// TIA Portal V20 export
ORGANIZATION_BLOCK "MainOB"   // OB126, LAD, ProgramCycle
TITLE = "Main Program Sweep (Cycle)"
{ S7_Optimized_Access := 'TRUE' }
// stored: SetENOAutomatically false
   VAR_INPUT
      Initial_Call : Bool;   // Initial call of this OB
      Remanence : Bool;   // =True, if remanent data are available
   END_VAR
   VAR_TEMP
      Temp : Bool;
   END_VAR
   VAR CONSTANT
      Constant_1 : Bool;
   END_VAR
BEGIN

REGION Network 1
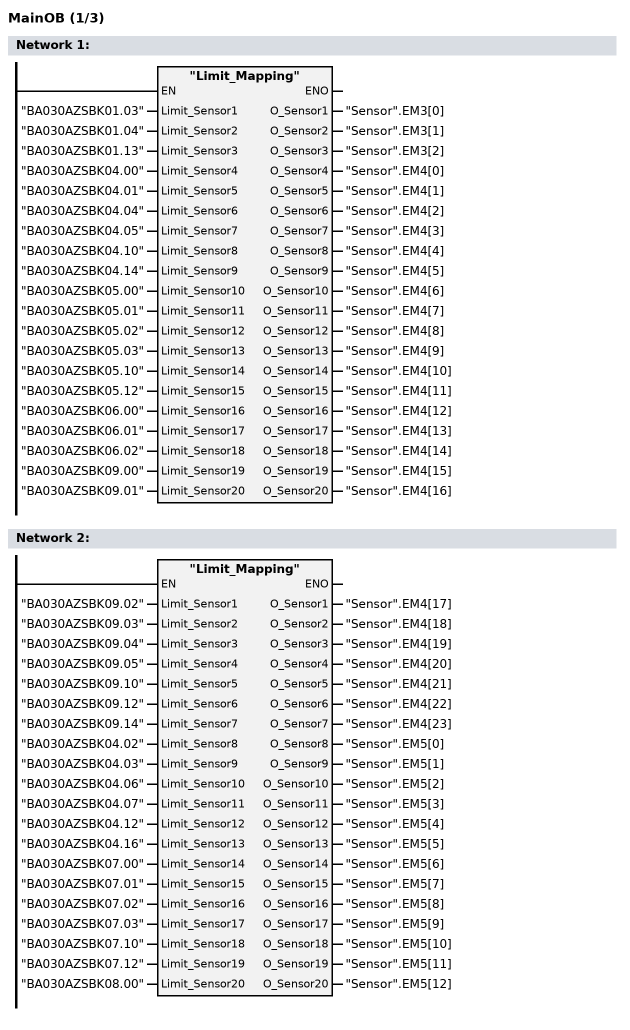
   RUNG wire#powerrail
      "Limit_Mapping"(Limit_Sensor1 := "BA030AZSBK01.03", Limit_Sensor2 := "BA030AZSBK01.04", Limit_Sensor3 := "BA030AZSBK01.13", Limit_Sensor4 := "BA030AZSBK04.00", Limit_Sensor5 := "BA030AZSBK04.01", Limit_Sensor6 := "BA030AZSBK04.04", Limit_Sensor7 := "BA030AZSBK04.05", Limit_Sensor8 := "BA030AZSBK04.10", Limit_Sensor9 := "BA030AZSBK04.14", Limit_Sensor10 := "BA030AZSBK05.00", Limit_Sensor11 := "BA030AZSBK05.01", Limit_Sensor12 := "BA030AZSBK05.02", Limit_Sensor13 := "BA030AZSBK05.03", Limit_Sensor14 := "BA030AZSBK05.10", Limit_Sensor15 := "BA030AZSBK05.12", Limit_Sensor16 := "BA030AZSBK06.00", Limit_Sensor17 := "BA030AZSBK06.01", Limit_Sensor18 := "BA030AZSBK06.02", Limit_Sensor19 := "BA030AZSBK09.00", Limit_Sensor20 := "BA030AZSBK09.01", O_Sensor1 => "Sensor".EM3[0], O_Sensor2 => "Sensor".EM3[1], O_Sensor3 => "Sensor".EM3[2], O_Sensor4 => "Sensor".EM4[0], O_Sensor5 => "Sensor".EM4[1], O_Sensor6 => "Sensor".EM4[2], O_Sensor7 => "Sensor".EM4[3], O_Sensor8 => "Sensor".EM4[4], O_Sensor9 => "Sensor".EM4[5], O_Sensor10 => "Sensor".EM4[6], O_Sensor11 => "Sensor".EM4[7], O_Sensor12 => "Sensor".EM4[8], O_Sensor13 => "Sensor".EM4[9], O_Sensor14 => "Sensor".EM4[10], O_Sensor15 => "Sensor".EM4[11], O_Sensor16 => "Sensor".EM4[12], O_Sensor17 => "Sensor".EM4[13], O_Sensor18 => "Sensor".EM4[14], O_Sensor19 => "Sensor".EM4[15], O_Sensor20 => "Sensor".EM4[16])
   END_RUNG
   // the same network as SCL:
   "Limit_Mapping"(Limit_Sensor1 := "BA030AZSBK01.03",
                   Limit_Sensor2 := "BA030AZSBK01.04",
                   Limit_Sensor3 := "BA030AZSBK01.13",
                   Limit_Sensor4 := "BA030AZSBK04.00",
                   Limit_Sensor5 := "BA030AZSBK04.01",
                   Limit_Sensor6 := "BA030AZSBK04.04",
                   Limit_Sensor7 := "BA030AZSBK04.05",
                   Limit_Sensor8 := "BA030AZSBK04.10",
                   Limit_Sensor9 := "BA030AZSBK04.14",
                   Limit_Sensor10 := "BA030AZSBK05.00",
                   Limit_Sensor11 := "BA030AZSBK05.01",
                   Limit_Sensor12 := "BA030AZSBK05.02",
                   Limit_Sensor13 := "BA030AZSBK05.03",
                   Limit_Sensor14 := "BA030AZSBK05.10",
                   Limit_Sensor15 := "BA030AZSBK05.12",
                   Limit_Sensor16 := "BA030AZSBK06.00",
                   Limit_Sensor17 := "BA030AZSBK06.01",
                   Limit_Sensor18 := "BA030AZSBK06.02",
                   Limit_Sensor19 := "BA030AZSBK09.00",
                   Limit_Sensor20 := "BA030AZSBK09.01",
                   O_Sensor1 => "Sensor".EM3[0],
                   O_Sensor2 => "Sensor".EM3[1],
                   O_Sensor3 => "Sensor".EM3[2],
                   O_Sensor4 => "Sensor".EM4[0],
                   O_Sensor5 => "Sensor".EM4[1],
                   O_Sensor6 => "Sensor".EM4[2],
                   O_Sensor7 => "Sensor".EM4[3],
                   O_Sensor8 => "Sensor".EM4[4],
                   O_Sensor9 => "Sensor".EM4[5],
                   O_Sensor10 => "Sensor".EM4[6],
                   O_Sensor11 => "Sensor".EM4[7],
                   O_Sensor12 => "Sensor".EM4[8],
                   O_Sensor13 => "Sensor".EM4[9],
                   O_Sensor14 => "Sensor".EM4[10],
                   O_Sensor15 => "Sensor".EM4[11],
                   O_Sensor16 => "Sensor".EM4[12],
                   O_Sensor17 => "Sensor".EM4[13],
                   O_Sensor18 => "Sensor".EM4[14],
                   O_Sensor19 => "Sensor".EM4[15],
                   O_Sensor20 => "Sensor".EM4[16]);
END_REGION

REGION Network 2
   RUNG wire#powerrail
      "Limit_Mapping"(Limit_Sensor1 := "BA030AZSBK09.02", Limit_Sensor2 := "BA030AZSBK09.03", Limit_Sensor3 := "BA030AZSBK09.04", Limit_Sensor4 := "BA030AZSBK09.05", Limit_Sensor5 := "BA030AZSBK09.10", Limit_Sensor6 := "BA030AZSBK09.12", Limit_Sensor7 := "BA030AZSBK09.14", Limit_Sensor8 := "BA030AZSBK04.02", Limit_Sensor9 := "BA030AZSBK04.03", Limit_Sensor10 := "BA030AZSBK04.06", Limit_Sensor11 := "BA030AZSBK04.07", Limit_Sensor12 := "BA030AZSBK04.12", Limit_Sensor13 := "BA030AZSBK04.16", Limit_Sensor14 := "BA030AZSBK07.00", Limit_Sensor15 := "BA030AZSBK07.01", Limit_Sensor16 := "BA030AZSBK07.02", Limit_Sensor17 := "BA030AZSBK07.03", Limit_Sensor18 := "BA030AZSBK07.10", Limit_Sensor19 := "BA030AZSBK07.12", Limit_Sensor20 := "BA030AZSBK08.00", O_Sensor1 => "Sensor".EM4[17], O_Sensor2 => "Sensor".EM4[18], O_Sensor3 => "Sensor".EM4[19], O_Sensor4 => "Sensor".EM4[20], O_Sensor5 => "Sensor".EM4[21], O_Sensor6 => "Sensor".EM4[22], O_Sensor7 => "Sensor".EM4[23], O_Sensor8 => "Sensor".EM5[0], O_Sensor9 => "Sensor".EM5[1], O_Sensor10 => "Sensor".EM5[2], O_Sensor11 => "Sensor".EM5[3], O_Sensor12 => "Sensor".EM5[4], O_Sensor13 => "Sensor".EM5[5], O_Sensor14 => "Sensor".EM5[6], O_Sensor15 => "Sensor".EM5[7], O_Sensor16 => "Sensor".EM5[8], O_Sensor17 => "Sensor".EM5[9], O_Sensor18 => "Sensor".EM5[10], O_Sensor19 => "Sensor".EM5[11], O_Sensor20 => "Sensor".EM5[12])
   END_RUNG
   // the same network as SCL:
   "Limit_Mapping"(Limit_Sensor1 := "BA030AZSBK09.02",
                   Limit_Sensor2 := "BA030AZSBK09.03",
                   Limit_Sensor3 := "BA030AZSBK09.04",
                   Limit_Sensor4 := "BA030AZSBK09.05",
                   Limit_Sensor5 := "BA030AZSBK09.10",
                   Limit_Sensor6 := "BA030AZSBK09.12",
                   Limit_Sensor7 := "BA030AZSBK09.14",
                   Limit_Sensor8 := "BA030AZSBK04.02",
                   Limit_Sensor9 := "BA030AZSBK04.03",
                   Limit_Sensor10 := "BA030AZSBK04.06",
                   Limit_Sensor11 := "BA030AZSBK04.07",
                   Limit_Sensor12 := "BA030AZSBK04.12",
                   Limit_Sensor13 := "BA030AZSBK04.16",
                   Limit_Sensor14 := "BA030AZSBK07.00",
                   Limit_Sensor15 := "BA030AZSBK07.01",
                   Limit_Sensor16 := "BA030AZSBK07.02",
                   Limit_Sensor17 := "BA030AZSBK07.03",
                   Limit_Sensor18 := "BA030AZSBK07.10",
                   Limit_Sensor19 := "BA030AZSBK07.12",
                   Limit_Sensor20 := "BA030AZSBK08.00",
                   O_Sensor1 => "Sensor".EM4[17],
                   O_Sensor2 => "Sensor".EM4[18],
                   O_Sensor3 => "Sensor".EM4[19],
                   O_Sensor4 => "Sensor".EM4[20],
                   O_Sensor5 => "Sensor".EM4[21],
                   O_Sensor6 => "Sensor".EM4[22],
                   O_Sensor7 => "Sensor".EM4[23],
                   O_Sensor8 => "Sensor".EM5[0],
                   O_Sensor9 => "Sensor".EM5[1],
                   O_Sensor10 => "Sensor".EM5[2],
                   O_Sensor11 => "Sensor".EM5[3],
                   O_Sensor12 => "Sensor".EM5[4],
                   O_Sensor13 => "Sensor".EM5[5],
                   O_Sensor14 => "Sensor".EM5[6],
                   O_Sensor15 => "Sensor".EM5[7],
                   O_Sensor16 => "Sensor".EM5[8],
                   O_Sensor17 => "Sensor".EM5[9],
                   O_Sensor18 => "Sensor".EM5[10],
                   O_Sensor19 => "Sensor".EM5[11],
                   O_Sensor20 => "Sensor".EM5[12]);
END_REGION

REGION Network 3
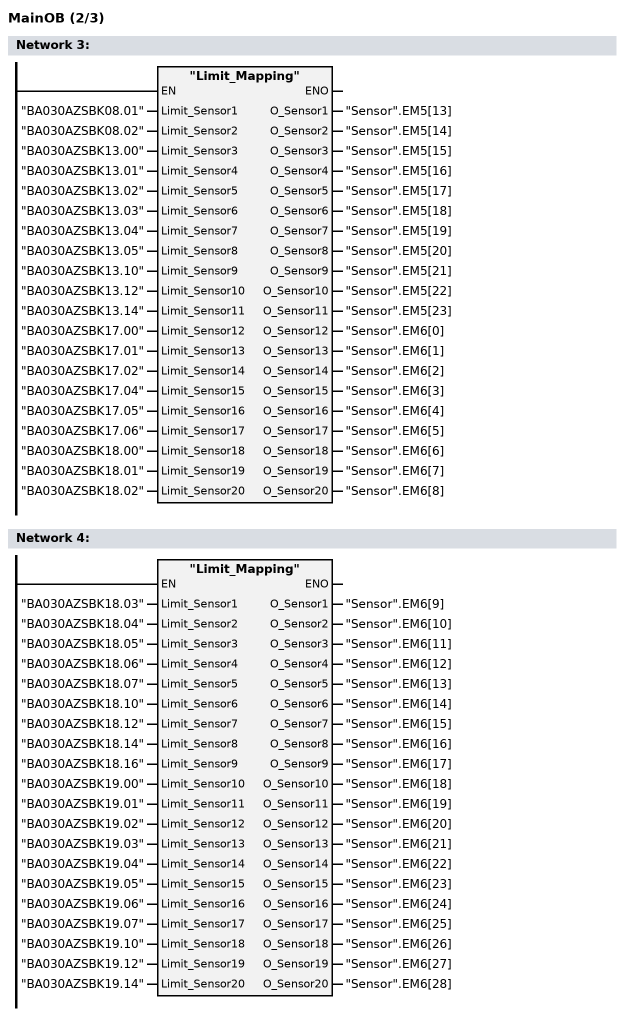
   RUNG wire#powerrail
      "Limit_Mapping"(Limit_Sensor1 := "BA030AZSBK08.01", Limit_Sensor2 := "BA030AZSBK08.02", Limit_Sensor3 := "BA030AZSBK13.00", Limit_Sensor4 := "BA030AZSBK13.01", Limit_Sensor5 := "BA030AZSBK13.02", Limit_Sensor6 := "BA030AZSBK13.03", Limit_Sensor7 := "BA030AZSBK13.04", Limit_Sensor8 := "BA030AZSBK13.05", Limit_Sensor9 := "BA030AZSBK13.10", Limit_Sensor10 := "BA030AZSBK13.12", Limit_Sensor11 := "BA030AZSBK13.14", Limit_Sensor12 := "BA030AZSBK17.00", Limit_Sensor13 := "BA030AZSBK17.01", Limit_Sensor14 := "BA030AZSBK17.02", Limit_Sensor15 := "BA030AZSBK17.04", Limit_Sensor16 := "BA030AZSBK17.05", Limit_Sensor17 := "BA030AZSBK17.06", Limit_Sensor18 := "BA030AZSBK18.00", Limit_Sensor19 := "BA030AZSBK18.01", Limit_Sensor20 := "BA030AZSBK18.02", O_Sensor1 => "Sensor".EM5[13], O_Sensor2 => "Sensor".EM5[14], O_Sensor3 => "Sensor".EM5[15], O_Sensor4 => "Sensor".EM5[16], O_Sensor5 => "Sensor".EM5[17], O_Sensor6 => "Sensor".EM5[18], O_Sensor7 => "Sensor".EM5[19], O_Sensor8 => "Sensor".EM5[20], O_Sensor9 => "Sensor".EM5[21], O_Sensor10 => "Sensor".EM5[22], O_Sensor11 => "Sensor".EM5[23], O_Sensor12 => "Sensor".EM6[0], O_Sensor13 => "Sensor".EM6[1], O_Sensor14 => "Sensor".EM6[2], O_Sensor15 => "Sensor".EM6[3], O_Sensor16 => "Sensor".EM6[4], O_Sensor17 => "Sensor".EM6[5], O_Sensor18 => "Sensor".EM6[6], O_Sensor19 => "Sensor".EM6[7], O_Sensor20 => "Sensor".EM6[8])
   END_RUNG
   // the same network as SCL:
   "Limit_Mapping"(Limit_Sensor1 := "BA030AZSBK08.01",
                   Limit_Sensor2 := "BA030AZSBK08.02",
                   Limit_Sensor3 := "BA030AZSBK13.00",
                   Limit_Sensor4 := "BA030AZSBK13.01",
                   Limit_Sensor5 := "BA030AZSBK13.02",
                   Limit_Sensor6 := "BA030AZSBK13.03",
                   Limit_Sensor7 := "BA030AZSBK13.04",
                   Limit_Sensor8 := "BA030AZSBK13.05",
                   Limit_Sensor9 := "BA030AZSBK13.10",
                   Limit_Sensor10 := "BA030AZSBK13.12",
                   Limit_Sensor11 := "BA030AZSBK13.14",
                   Limit_Sensor12 := "BA030AZSBK17.00",
                   Limit_Sensor13 := "BA030AZSBK17.01",
                   Limit_Sensor14 := "BA030AZSBK17.02",
                   Limit_Sensor15 := "BA030AZSBK17.04",
                   Limit_Sensor16 := "BA030AZSBK17.05",
                   Limit_Sensor17 := "BA030AZSBK17.06",
                   Limit_Sensor18 := "BA030AZSBK18.00",
                   Limit_Sensor19 := "BA030AZSBK18.01",
                   Limit_Sensor20 := "BA030AZSBK18.02",
                   O_Sensor1 => "Sensor".EM5[13],
                   O_Sensor2 => "Sensor".EM5[14],
                   O_Sensor3 => "Sensor".EM5[15],
                   O_Sensor4 => "Sensor".EM5[16],
                   O_Sensor5 => "Sensor".EM5[17],
                   O_Sensor6 => "Sensor".EM5[18],
                   O_Sensor7 => "Sensor".EM5[19],
                   O_Sensor8 => "Sensor".EM5[20],
                   O_Sensor9 => "Sensor".EM5[21],
                   O_Sensor10 => "Sensor".EM5[22],
                   O_Sensor11 => "Sensor".EM5[23],
                   O_Sensor12 => "Sensor".EM6[0],
                   O_Sensor13 => "Sensor".EM6[1],
                   O_Sensor14 => "Sensor".EM6[2],
                   O_Sensor15 => "Sensor".EM6[3],
                   O_Sensor16 => "Sensor".EM6[4],
                   O_Sensor17 => "Sensor".EM6[5],
                   O_Sensor18 => "Sensor".EM6[6],
                   O_Sensor19 => "Sensor".EM6[7],
                   O_Sensor20 => "Sensor".EM6[8]);
END_REGION

REGION Network 4
   RUNG wire#powerrail
      "Limit_Mapping"(Limit_Sensor1 := "BA030AZSBK18.03", Limit_Sensor2 := "BA030AZSBK18.04", Limit_Sensor3 := "BA030AZSBK18.05", Limit_Sensor4 := "BA030AZSBK18.06", Limit_Sensor5 := "BA030AZSBK18.07", Limit_Sensor6 := "BA030AZSBK18.10", Limit_Sensor7 := "BA030AZSBK18.12", Limit_Sensor8 := "BA030AZSBK18.14", Limit_Sensor9 := "BA030AZSBK18.16", Limit_Sensor10 := "BA030AZSBK19.00", Limit_Sensor11 := "BA030AZSBK19.01", Limit_Sensor12 := "BA030AZSBK19.02", Limit_Sensor13 := "BA030AZSBK19.03", Limit_Sensor14 := "BA030AZSBK19.04", Limit_Sensor15 := "BA030AZSBK19.05", Limit_Sensor16 := "BA030AZSBK19.06", Limit_Sensor17 := "BA030AZSBK19.07", Limit_Sensor18 := "BA030AZSBK19.10", Limit_Sensor19 := "BA030AZSBK19.12", Limit_Sensor20 := "BA030AZSBK19.14", O_Sensor1 => "Sensor".EM6[9], O_Sensor2 => "Sensor".EM6[10], O_Sensor3 => "Sensor".EM6[11], O_Sensor4 => "Sensor".EM6[12], O_Sensor5 => "Sensor".EM6[13], O_Sensor6 => "Sensor".EM6[14], O_Sensor7 => "Sensor".EM6[15], O_Sensor8 => "Sensor".EM6[16], O_Sensor9 => "Sensor".EM6[17], O_Sensor10 => "Sensor".EM6[18], O_Sensor11 => "Sensor".EM6[19], O_Sensor12 => "Sensor".EM6[20], O_Sensor13 => "Sensor".EM6[21], O_Sensor14 => "Sensor".EM6[22], O_Sensor15 => "Sensor".EM6[23], O_Sensor16 => "Sensor".EM6[24], O_Sensor17 => "Sensor".EM6[25], O_Sensor18 => "Sensor".EM6[26], O_Sensor19 => "Sensor".EM6[27], O_Sensor20 => "Sensor".EM6[28])
   END_RUNG
   // the same network as SCL:
   "Limit_Mapping"(Limit_Sensor1 := "BA030AZSBK18.03",
                   Limit_Sensor2 := "BA030AZSBK18.04",
                   Limit_Sensor3 := "BA030AZSBK18.05",
                   Limit_Sensor4 := "BA030AZSBK18.06",
                   Limit_Sensor5 := "BA030AZSBK18.07",
                   Limit_Sensor6 := "BA030AZSBK18.10",
                   Limit_Sensor7 := "BA030AZSBK18.12",
                   Limit_Sensor8 := "BA030AZSBK18.14",
                   Limit_Sensor9 := "BA030AZSBK18.16",
                   Limit_Sensor10 := "BA030AZSBK19.00",
                   Limit_Sensor11 := "BA030AZSBK19.01",
                   Limit_Sensor12 := "BA030AZSBK19.02",
                   Limit_Sensor13 := "BA030AZSBK19.03",
                   Limit_Sensor14 := "BA030AZSBK19.04",
                   Limit_Sensor15 := "BA030AZSBK19.05",
                   Limit_Sensor16 := "BA030AZSBK19.06",
                   Limit_Sensor17 := "BA030AZSBK19.07",
                   Limit_Sensor18 := "BA030AZSBK19.10",
                   Limit_Sensor19 := "BA030AZSBK19.12",
                   Limit_Sensor20 := "BA030AZSBK19.14",
                   O_Sensor1 => "Sensor".EM6[9],
                   O_Sensor2 => "Sensor".EM6[10],
                   O_Sensor3 => "Sensor".EM6[11],
                   O_Sensor4 => "Sensor".EM6[12],
                   O_Sensor5 => "Sensor".EM6[13],
                   O_Sensor6 => "Sensor".EM6[14],
                   O_Sensor7 => "Sensor".EM6[15],
                   O_Sensor8 => "Sensor".EM6[16],
                   O_Sensor9 => "Sensor".EM6[17],
                   O_Sensor10 => "Sensor".EM6[18],
                   O_Sensor11 => "Sensor".EM6[19],
                   O_Sensor12 => "Sensor".EM6[20],
                   O_Sensor13 => "Sensor".EM6[21],
                   O_Sensor14 => "Sensor".EM6[22],
                   O_Sensor15 => "Sensor".EM6[23],
                   O_Sensor16 => "Sensor".EM6[24],
                   O_Sensor17 => "Sensor".EM6[25],
                   O_Sensor18 => "Sensor".EM6[26],
                   O_Sensor19 => "Sensor".EM6[27],
                   O_Sensor20 => "Sensor".EM6[28]);
END_REGION

REGION Network 5
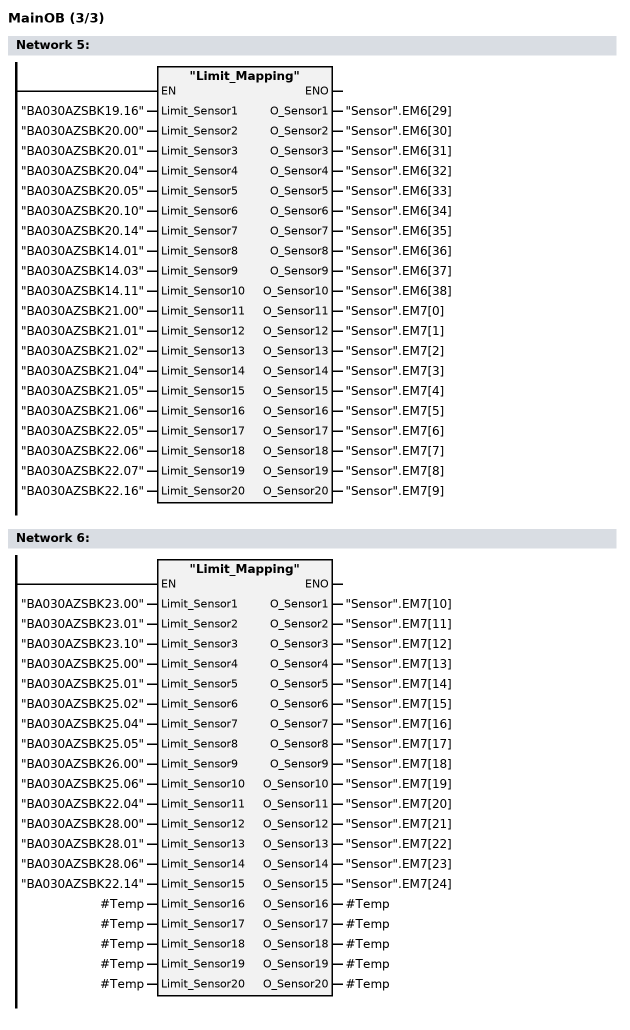
   RUNG wire#powerrail
      "Limit_Mapping"(Limit_Sensor1 := "BA030AZSBK19.16", Limit_Sensor2 := "BA030AZSBK20.00", Limit_Sensor3 := "BA030AZSBK20.01", Limit_Sensor4 := "BA030AZSBK20.04", Limit_Sensor5 := "BA030AZSBK20.05", Limit_Sensor6 := "BA030AZSBK20.10", Limit_Sensor7 := "BA030AZSBK20.14", Limit_Sensor8 := "BA030AZSBK14.01", Limit_Sensor9 := "BA030AZSBK14.03", Limit_Sensor10 := "BA030AZSBK14.11", Limit_Sensor11 := "BA030AZSBK21.00", Limit_Sensor12 := "BA030AZSBK21.01", Limit_Sensor13 := "BA030AZSBK21.02", Limit_Sensor14 := "BA030AZSBK21.04", Limit_Sensor15 := "BA030AZSBK21.05", Limit_Sensor16 := "BA030AZSBK21.06", Limit_Sensor17 := "BA030AZSBK22.05", Limit_Sensor18 := "BA030AZSBK22.06", Limit_Sensor19 := "BA030AZSBK22.07", Limit_Sensor20 := "BA030AZSBK22.16", O_Sensor1 => "Sensor".EM6[29], O_Sensor2 => "Sensor".EM6[30], O_Sensor3 => "Sensor".EM6[31], O_Sensor4 => "Sensor".EM6[32], O_Sensor5 => "Sensor".EM6[33], O_Sensor6 => "Sensor".EM6[34], O_Sensor7 => "Sensor".EM6[35], O_Sensor8 => "Sensor".EM6[36], O_Sensor9 => "Sensor".EM6[37], O_Sensor10 => "Sensor".EM6[38], O_Sensor11 => "Sensor".EM7[0], O_Sensor12 => "Sensor".EM7[1], O_Sensor13 => "Sensor".EM7[2], O_Sensor14 => "Sensor".EM7[3], O_Sensor15 => "Sensor".EM7[4], O_Sensor16 => "Sensor".EM7[5], O_Sensor17 => "Sensor".EM7[6], O_Sensor18 => "Sensor".EM7[7], O_Sensor19 => "Sensor".EM7[8], O_Sensor20 => "Sensor".EM7[9])
   END_RUNG
   // the same network as SCL:
   "Limit_Mapping"(Limit_Sensor1 := "BA030AZSBK19.16",
                   Limit_Sensor2 := "BA030AZSBK20.00",
                   Limit_Sensor3 := "BA030AZSBK20.01",
                   Limit_Sensor4 := "BA030AZSBK20.04",
                   Limit_Sensor5 := "BA030AZSBK20.05",
                   Limit_Sensor6 := "BA030AZSBK20.10",
                   Limit_Sensor7 := "BA030AZSBK20.14",
                   Limit_Sensor8 := "BA030AZSBK14.01",
                   Limit_Sensor9 := "BA030AZSBK14.03",
                   Limit_Sensor10 := "BA030AZSBK14.11",
                   Limit_Sensor11 := "BA030AZSBK21.00",
                   Limit_Sensor12 := "BA030AZSBK21.01",
                   Limit_Sensor13 := "BA030AZSBK21.02",
                   Limit_Sensor14 := "BA030AZSBK21.04",
                   Limit_Sensor15 := "BA030AZSBK21.05",
                   Limit_Sensor16 := "BA030AZSBK21.06",
                   Limit_Sensor17 := "BA030AZSBK22.05",
                   Limit_Sensor18 := "BA030AZSBK22.06",
                   Limit_Sensor19 := "BA030AZSBK22.07",
                   Limit_Sensor20 := "BA030AZSBK22.16",
                   O_Sensor1 => "Sensor".EM6[29],
                   O_Sensor2 => "Sensor".EM6[30],
                   O_Sensor3 => "Sensor".EM6[31],
                   O_Sensor4 => "Sensor".EM6[32],
                   O_Sensor5 => "Sensor".EM6[33],
                   O_Sensor6 => "Sensor".EM6[34],
                   O_Sensor7 => "Sensor".EM6[35],
                   O_Sensor8 => "Sensor".EM6[36],
                   O_Sensor9 => "Sensor".EM6[37],
                   O_Sensor10 => "Sensor".EM6[38],
                   O_Sensor11 => "Sensor".EM7[0],
                   O_Sensor12 => "Sensor".EM7[1],
                   O_Sensor13 => "Sensor".EM7[2],
                   O_Sensor14 => "Sensor".EM7[3],
                   O_Sensor15 => "Sensor".EM7[4],
                   O_Sensor16 => "Sensor".EM7[5],
                   O_Sensor17 => "Sensor".EM7[6],
                   O_Sensor18 => "Sensor".EM7[7],
                   O_Sensor19 => "Sensor".EM7[8],
                   O_Sensor20 => "Sensor".EM7[9]);
END_REGION

REGION Network 6
   RUNG wire#powerrail
      "Limit_Mapping"(Limit_Sensor1 := "BA030AZSBK23.00", Limit_Sensor2 := "BA030AZSBK23.01", Limit_Sensor3 := "BA030AZSBK23.10", Limit_Sensor4 := "BA030AZSBK25.00", Limit_Sensor5 := "BA030AZSBK25.01", Limit_Sensor6 := "BA030AZSBK25.02", Limit_Sensor7 := "BA030AZSBK25.04", Limit_Sensor8 := "BA030AZSBK25.05", Limit_Sensor9 := "BA030AZSBK26.00", Limit_Sensor10 := "BA030AZSBK25.06", Limit_Sensor11 := "BA030AZSBK22.04", Limit_Sensor12 := "BA030AZSBK28.00", Limit_Sensor13 := "BA030AZSBK28.01", Limit_Sensor14 := "BA030AZSBK28.06", Limit_Sensor15 := "BA030AZSBK22.14", Limit_Sensor16 := #Temp, Limit_Sensor17 := #Temp, Limit_Sensor18 := #Temp, Limit_Sensor19 := #Temp, Limit_Sensor20 := #Temp, O_Sensor1 => "Sensor".EM7[10], O_Sensor2 => "Sensor".EM7[11], O_Sensor3 => "Sensor".EM7[12], O_Sensor4 => "Sensor".EM7[13], O_Sensor5 => "Sensor".EM7[14], O_Sensor6 => "Sensor".EM7[15], O_Sensor7 => "Sensor".EM7[16], O_Sensor8 => "Sensor".EM7[17], O_Sensor9 => "Sensor".EM7[18], O_Sensor10 => "Sensor".EM7[19], O_Sensor11 => "Sensor".EM7[20], O_Sensor12 => "Sensor".EM7[21], O_Sensor13 => "Sensor".EM7[22], O_Sensor14 => "Sensor".EM7[23], O_Sensor15 => "Sensor".EM7[24], O_Sensor16 => #Temp, O_Sensor17 => #Temp, O_Sensor18 => #Temp, O_Sensor19 => #Temp, O_Sensor20 => #Temp)
   END_RUNG
   // the same network as SCL:
   "Limit_Mapping"(Limit_Sensor1 := "BA030AZSBK23.00",
                   Limit_Sensor2 := "BA030AZSBK23.01",
                   Limit_Sensor3 := "BA030AZSBK23.10",
                   Limit_Sensor4 := "BA030AZSBK25.00",
                   Limit_Sensor5 := "BA030AZSBK25.01",
                   Limit_Sensor6 := "BA030AZSBK25.02",
                   Limit_Sensor7 := "BA030AZSBK25.04",
                   Limit_Sensor8 := "BA030AZSBK25.05",
                   Limit_Sensor9 := "BA030AZSBK26.00",
                   Limit_Sensor10 := "BA030AZSBK25.06",
                   Limit_Sensor11 := "BA030AZSBK22.04",
                   Limit_Sensor12 := "BA030AZSBK28.00",
                   Limit_Sensor13 := "BA030AZSBK28.01",
                   Limit_Sensor14 := "BA030AZSBK28.06",
                   Limit_Sensor15 := "BA030AZSBK22.14",
                   Limit_Sensor16 := #Temp,
                   Limit_Sensor17 := #Temp,
                   Limit_Sensor18 := #Temp,
                   Limit_Sensor19 := #Temp,
                   Limit_Sensor20 := #Temp,
                   O_Sensor1 => "Sensor".EM7[10],
                   O_Sensor2 => "Sensor".EM7[11],
                   O_Sensor3 => "Sensor".EM7[12],
                   O_Sensor4 => "Sensor".EM7[13],
                   O_Sensor5 => "Sensor".EM7[14],
                   O_Sensor6 => "Sensor".EM7[15],
                   O_Sensor7 => "Sensor".EM7[16],
                   O_Sensor8 => "Sensor".EM7[17],
                   O_Sensor9 => "Sensor".EM7[18],
                   O_Sensor10 => "Sensor".EM7[19],
                   O_Sensor11 => "Sensor".EM7[20],
                   O_Sensor12 => "Sensor".EM7[21],
                   O_Sensor13 => "Sensor".EM7[22],
                   O_Sensor14 => "Sensor".EM7[23],
                   O_Sensor15 => "Sensor".EM7[24],
                   O_Sensor16 => #Temp,
                   O_Sensor17 => #Temp,
                   O_Sensor18 => #Temp,
                   O_Sensor19 => #Temp,
                   O_Sensor20 => #Temp);
END_REGION
END_ORGANIZATION_BLOCK
